{attribute 'enable_dynamic_creation'}
FUNCTION_BLOCK FB_CondiStepResult EXTENDS FB_CondiBase
VAR_INPUT
END_VAR
VAR_OUTPUT
END_VAR
VAR
	pStep 			: POINTER TO ST_Step;
	eCompareOperator: E_CompOperator;
	nCompareValue 	: DINT;
END_VAR

PROPERTY P_eCompareOperator : E_CompOperator
GET
P_eCompareOperator := eCompareOperator;
END_GET
SET
eCompareOperator := P_eCompareOperator;
END_SET
END_PROPERTY

PROPERTY P_nCompareValue : DINT
SET
nCompareValue := P_nCompareValue;
END_SET
END_PROPERTY

PROPERTY P_pStep : POINTER TO ST_Step
SET
pStep := P_pStep;
END_SET
END_PROPERTY

METHOD M_Check : BYTE
VAR_INPUT
	nPreResult : BYTE;
END_VAR

VAR
	bCancel : BOOL := TRUE;
END_VAR
IF pStep^.bActionResultIsValid  AND (pStep^.eState = E_StepState.STEPSTATUS_Ready) THEN
	IF eCondiOperator = E_LogicOperator.LOGIC_OP_AND THEN
		//nPreResult.0 := nPreResult.0 AND TRUE;
	ELSIF eCondiOperator = E_LogicOperator.LOGIC_OP_OR THEN
		nPreResult.0 := TRUE;
	END_IF
	
	IF nPreResult.0 THEN
		CASE eCompareOperator OF
			E_CompOperator.COMP_OP_GT:	//>
				IF pStep^.nActionResult > nCompareValue THEN
					bCancel := FALSE;
				END_IF
			E_CompOperator.COMP_OP_LT:	//<
				IF pStep^.nActionResult < nCompareValue THEN
					bCancel := FALSE;
				END_IF
			E_CompOperator.COMP_OP_GE:	//>=
				IF pStep^.nActionResult >= nCompareValue THEN
					bCancel := FALSE;
				END_IF
			E_CompOperator.COMP_OP_LE:	//<=
				IF pStep^.nActionResult <= nCompareValue THEN
					bCancel := FALSE;
				END_IF
			E_CompOperator.COMP_OP_EQ:	//=
				IF pStep^.nActionResult = nCompareValue THEN
					bCancel := FALSE;
				END_IF
		END_CASE
		
		IF eCondiOperator = E_LogicOperator.LOGIC_OP_AND THEN
			nPreResult.1 := nPreResult.1 OR bCancel;
		ELSIF eCondiOperator = E_LogicOperator.LOGIC_OP_OR THEN
			IF NOT bCancel THEN
				nPreResult.1 := FALSE;
			END_IF
		END_IF
		
		IF pNextCondi > 0 THEN
			M_Check := pNextCondi^.M_Check(nPreResult);
		ELSE
			M_Check  := nPreResult;
		END_IF		
	END_IF
END_IF
END_METHOD

END_FUNCTION_BLOCK

(* stored: Version 1.1.0.1, ProductVersion 3.1.4022.10
   POU FB_CondiStepResult: Id {72836e5d-189d-419c-a7fd-efb986e596ad}, SpecialFunc None
   Property P_eCompareOperator: Id {01e4eb2e-4ebd-49f8-9c96-36348f2f11fd}
   Get Get: Id {b5554202-0145-4935-9c7c-93a41057725b}
   Set Set: Id {d2e1a7df-8439-483c-8fbf-2bce565c94e2}
   Property P_nCompareValue: Id {492692de-1d2c-47a5-a0ad-fbad52f74397}
   Set Set: Id {6edb6f2c-b153-4c19-a139-8498ada3aca2}
   Property P_pStep: Id {7131c9bb-5ac9-4915-a879-4b11ba685acc}
   Set Set: Id {10c0986e-60cf-4405-9699-b992f9151ebd}
   Method M_Check: Id {8c010451-2980-4e58-ba1a-1ba29afe414b} *)
